{attribute 'linkalways'} 
{attribute 'no_explicit_call' := 'This FB is a CLASS and must be accessed using methods or properties'}
{attribute 'enable_dynamic_creation'}
FUNCTION_BLOCK FINAL ABS_BYTE EXTENDS Node
VAR
	in : _BYTE(0);
	out : _BYTE(0);
END_VAR

METHOD PUBLIC Clone : I_Node
VAR
	pNode : POINTER TO ABS_BYTE;
END_VAR
pNode := __NEW(ABS_BYTE);
Clone := pNode^;
END_METHOD

METHOD FB_init : BOOL
VAR_INPUT
	bInitRetains : BOOL; // if TRUE, the retain variables are initialized (warm start / cold start)
	bInCopyCode : BOOL;  // if TRUE, the instance afterwards gets moved into the copy code (online change)
END_VAR
AddInput('in',THIS^.in);
AddOutput('out', THIS^.out);
END_METHOD

METHOD PROTECTED OnExecute
VAR
END_VAR
out.Value := ABS(in.Value);
END_METHOD

END_FUNCTION_BLOCK

(* stored: Version 1.1.0.1, ProductVersion 3.1.4024.15
   POU ABS_BYTE: Id {a287964e-085f-4bf1-a871-b9885872cfb9}, SpecialFunc None
   Folder Constructor: Id {7ff4a368-7b4f-4b69-a71e-93b3156ae2d6}
   Method Clone: Id {f4ff4a41-19bf-44f7-8e09-3825f5bb5a77}
   Method FB_init: Id {33309d64-ab7e-46eb-9051-76563b8b0867}
   Method OnExecute: Id {febe98b9-110f-43af-8edb-61c2de5f1a55} *)
